(*
:Beskrivning:	| Läser systemtiden.
:Instruktioner:	| Ändra sAMSNetID för annan tidsserver. Lämna tom för lokal tid i PLC.

:Versionshistorik:
+-------------+------------+----------------+------------+------------------------------------------+
|Datum        | Version    | Skapad under   | Författare | Kommentar                                |
+=============+============+================+============+==========================================+
|2020-02-20   | 1.0.0.1    | V3.1.4022.30   | CMC dev.   | Funktionsblock skapat                    |
+-------------+------------+----------------+------------+------------------------------------------+
	
*)
FUNCTION_BLOCK FB_SystemTime
VAR_INPUT
	sAMSNetID			: STRING:='';	// AMSNet-ID
END_VAR

VAR_OUTPUT
	dtSystemTime		: DT;			// Systemtid
	bGetTimeBusy		: BOOL;			// Busy  		
	bGetTimeError		: BOOL;			// Error
	nGetTimeErrorCode	: UDINT;		// ErrorID
	nYear				: DWORD;		// År
	nMonth				: DWORD;		// Månad
	nDay				: DWORD;		// Dag
	nWeekDay 			: DWORD;		// Veckodag
	nHour				: DWORD;		// Timme
	nMinute 			: DWORD;		// Minut
	nSecond				: DWORD;		// Sekund
	nMilliSecond		: DWORD;		// Millisekund
	nHourMinute			: DWORD;		// Timme och minut (HHMM)
END_VAR

VAR
	fbGetTime			: NT_GetTime;
	fbTimerPulseSec		: FB_TimerPulseSec;
END_VAR

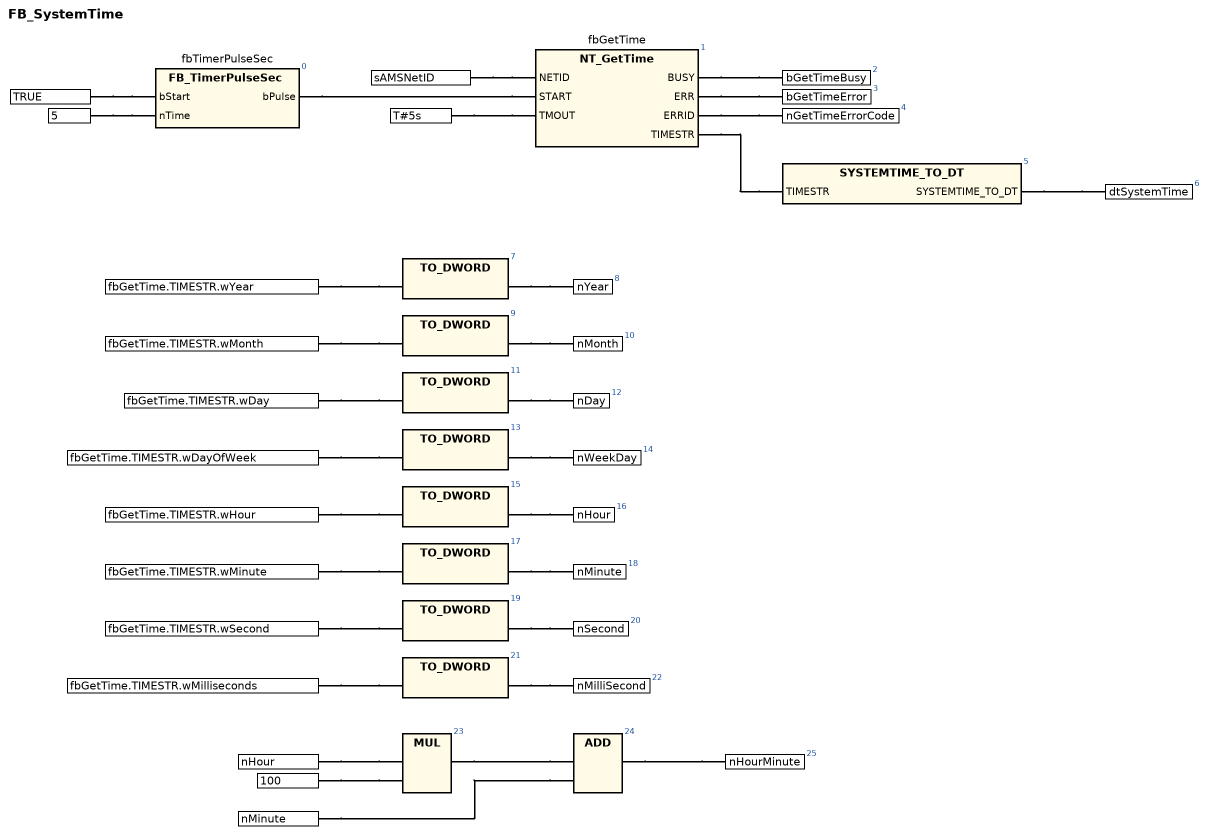
fbTimerPulseSec(bStart := TRUE, nTime := 5); // FB_TimerPulseSec
fbGetTime(NETID := sAMSNetID, START := fbTimerPulseSec.bPulse, TMOUT := T#5s); // NT_GetTime
bGetTimeBusy := fbGetTime.BUSY;
bGetTimeError := fbGetTime.ERR;
nGetTimeErrorCode := fbGetTime.ERRID;
dtSystemTime := SYSTEMTIME_TO_DT(TIMESTR := fbGetTime.TIMESTR);
nYear := TO_DWORD(fbGetTime.TIMESTR.wYear);
nMonth := TO_DWORD(fbGetTime.TIMESTR.wMonth);
nDay := TO_DWORD(fbGetTime.TIMESTR.wDay);
nWeekDay := TO_DWORD(fbGetTime.TIMESTR.wDayOfWeek);
nHour := TO_DWORD(fbGetTime.TIMESTR.wHour);
nMinute := TO_DWORD(fbGetTime.TIMESTR.wMinute);
nSecond := TO_DWORD(fbGetTime.TIMESTR.wSecond);
nMilliSecond := TO_DWORD(fbGetTime.TIMESTR.wMilliseconds);
nHourMinute := nHour * 100 + nMinute;

END_FUNCTION_BLOCK

(* stored: Version 1.1.0.1, ProductVersion 3.1.4024.11
   POU FB_SystemTime: Id {bfefd999-c78c-4384-b542-af89599aa214}, SpecialFunc None *)
